Staubli VAL3: takestop.pgx

program takestop()
begin
  //
  while true
    if distop==true
      bstop=true
    endIf
    if distart==true
      bstop=false
    endIf
    delay(0)
  endWhile
end
